// SIMATIC STEP 7 (V5.x) project plc
// CPU: CPU 315-2DP
// station: 硬件
// station: SIMATIC 300(1)
// station: P_ADR_BUS
// program: S7 程序(1)

DATA_BLOCK DB 1
VERSION : 0.1
  STRUCT
   dd : INT ;	//临时占位符变量
   cc : INT ;
  END_STRUCT ;	
BEGIN
END_DATA_BLOCK

ORGANIZATION_BLOCK OB 1
TITLE = "Main Program Sweep (Cycle)"
VERSION : 0.1
VAR_TEMP
  OB1_EV_CLASS : BYTE ;	//Bits 0-3 = 1 (Coming event), Bits 4-7 = 1 (Event class 1)
  OB1_SCAN_1 : BYTE ;	//1 (Cold restart scan 1 of OB 1), 3 (Scan 2-n of OB 1)
  OB1_PRIORITY : BYTE ;	//Priority of OB Execution
  OB1_OB_NUMBR : BYTE ;	//1 (Organization block 1, OB1)
  OB1_RESERVED_1 : BYTE ;	//Reserved for system
  OB1_RESERVED_2 : BYTE ;	//Reserved for system
  OB1_PREV_CYCLE : INT ;	//Cycle time of previous OB1 scan (milliseconds)
  OB1_MIN_CYCLE : INT ;	//Minimum cycle time of OB1 (milliseconds)
  OB1_MAX_CYCLE : INT ;	//Maximum cycle time of OB1 (milliseconds)
  OB1_DATE_TIME : DATE_AND_TIME ;	//Date and time OB1 started
END_VAR
BEGIN
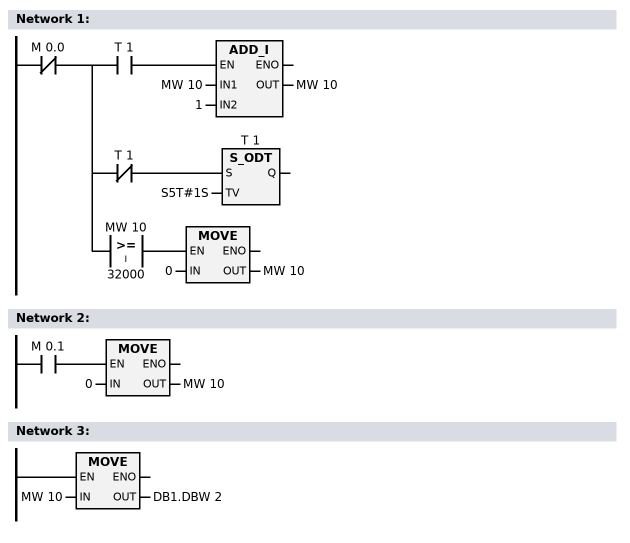
NETWORK
TITLE =
      AN    M 0.0;
      =     L 20.0;
      A     L 20.0;
      A     T 1;
      JNB   _001;
      L     MW 10;
      L     1;
      +I;
      T     MW 10;
_001: NOP   0;
      A     L 20.0;
      AN    T 1;
      L     S5T#1S;
      SD    T 1;
      NOP   0;
      NOP   0;
      NOP   0;
      NOP   0;
      A     L 20.0;
      A(;
      L     MW 10;
      L     32000;
      >=I;
      );
      JNB   _002;
      L     0;
      T     MW 10;
_002: NOP   0;
NETWORK
TITLE =
      A     M 0.1;
      JNB   _003;
      L     0;
      T     MW 10;
_003: NOP   0;
NETWORK
TITLE =
      L     MW 10;
      T     DB1.DBW 2;
      NOP   0;
END_ORGANIZATION_BLOCK
